TYPE st_recipe_titles :
	STRUCT
		pusher					:STRING;
		compress				:STRING;
		shield					:STRING;
		clamp					:STRING;
		offset					:STRING;
		
	END_STRUCT
END_TYPE

(* stored: Version 1.1.0.1, ProductVersion 3.1.4020.12
   DUT st_recipe_titles: Id {4441526d-c07f-4a00-9bc6-8fc215be5d72} *)
